// TIA Portal V20 export
DATA_BLOCK "PM9"   // DB283
// stored: MemoryReserve 100
   VAR
      "FINAL VISION STAGE LIFT UP" : Bool;
      "FINAL VISION STAGE LIFT DOWN" : Bool;
      "FINAL VISION LIGHT UP" : Bool;
      "FINAL VISION LIGHT DOWN" : Bool;
      "LASER MARKING COVER UP" : Bool;
      "LASER MARKING COVER DOWN" : Bool;
      "LASER MARKING STAGE LIFT UP" : Bool;
      "LASER MARKING STAGE LIFT DOWN" : Bool;
      SPARE : Bool;
      SPARE_1 : Bool;
      "INS TRANSFER P&P CLAMP #1 CLOSE" : Bool;
      "INS TRANSFER P&P CLAMP #1 OPEN" : Bool;
      "INS TRANSFER P&P CLAMP #2 CLOSE" : Bool;
      "INS TRANSFER P&P CLAMP #2 OPEN" : Bool;
      "JR Unloading P&P CLAMP CLOSE" : Bool;
      "JR Unloading P&P CLAMP OPEN" : Bool;
   END_VAR
BEGIN
END_DATA_BLOCK
